FUNCTION TryConvert_DWORD_TO_SINT : BOOL
VAR_INPUT
	in : DWORD;
	out : REFERENCE TO SINT;
END_VAR

IF in > DatatypeLimits.MAX_VALUE_OF_DWORD_WHICH_CAN_BE_HELD_IN_A_SINT THEN
	RETURN;
END_IF

out := DWORD_TO_SINT(in);
TryConvert_DWORD_TO_SINT := TRUE;

END_FUNCTION

(* stored: Version 1.1.0.1, ProductVersion 3.1.4024.12
   POU TryConvert_DWORD_TO_SINT: Id {ce5c5ed0-5c0f-4f3e-b7cd-9b6ae5ea7522}, SpecialFunc None *)
